# EPICS autosave request: iocBoot/ioc13laser/auto_positions.req
file "CARS_8_motor_positions.req",       P=$(P)
~
